// TIA Portal V17 export
// export: Created 2026-04-13T11:12:42.4906575Z, ExportSetting WithDefaults, DisplayName Totally Integrated Automation Portal, DisplayVersion V17 Update 4, DisplayName TIA Portal Openness, DisplayVersion V17 Update 4, DisplayName TIA Portal Version Control Interface, DisplayVersion V17, DisplayName SINAMICS Startdrive Advanced, DisplayVersion V17, DisplayName SINAMICS Startdrive G130, G150, S120, S150, SINAMICS MV, S210, DisplayVersion V17, DisplayName SINAMICS Startdrive G110M, G120, G120C, G120D, G120P, G115D, DisplayVersion V17, DisplayName STEP 7 Professional, DisplayVersion V17 Update 4, DisplayName STEP 7 Safety, DisplayVersion V17, DisplayName WinCC Professional, DisplayVersion V17 Update 4
FUNCTION_BLOCK "5-称重法堵塞"   // FB76, LAD
{ S7_Optimized_Access := 'TRUE' }
VERSION : 0.1
// stored: AutoNumber true, IsIECCheckEnabled false, IsRetainMemResEnabled false, MemoryReserve 100, SetENOAutomatically false, UDAEnableTagReadback false
   VAR_OUTPUT
      进料堵塞辅助 : Bool;
   END_VAR
   VAR_IN_OUT
      进料蠕动泵开关 : Bool;
      当前重量值 : Real;
      上一次重量值 : Real;
      重量差值 : Real;
      称重仪实际重量 : Real;
      设定物料检测重量 : Real;
   END_VAR
BEGIN

REGION Network 1 (SCL): 初扫描 / 油炉和风机
   // 需放入Cyclic interrupt中，并设置间隔时间60000ms
   #当前重量值 := #称重仪实际重量;
   #重量差值 := #当前重量值 - #上一次重量值;
   #上一次重量值 := #称重仪实际重量;

   IF #进料蠕动泵开关 AND #重量差值 <= #设定物料检测重量 THEN
       #进料堵塞辅助 := true;
   END_IF;
END_REGION
END_FUNCTION_BLOCK
